(* CODESYS project twincat-tools.library
   Company: hganchev
   DefaultNamespace: tc-tools
   Version: 1.0.0.0
   DocFormat: reStructuredText
   Placeholder: tc-tools
   Author: hganchev
   Title: tc-tools

Project tree, tasks and I/O mapping:
  libraries: Tc2_Standard, * (Beckhoff Automation GmbH); Tc2_System, * (Beckhoff Automation GmbH); Tc2_Utilities, * (Beckhoff Automation GmbH); Tc3_Module, * (Beckhoff Automation GmbH); Tc2_MC2, * (Beckhoff Automation GmbH)
  DUTs/
  GVLs/
    global variables Parameters
  POUs/
    AxisControl/
      function block MC_AxisControl [ST]
    Export/
      function block ExportArrayREALDataToTextFile [ST]
    Range/
      function F_GET_IN_RANGE_INT [ST]
      function F_IN_BOUNDS_ARRAY_INT [ST]
    Round/
      function F_ROUND_LREAL [ST]
      function F_ROUND_REAL [ST]
    String/
      function F_STRING_SPLIT [ST]
    TimeStamp/
      function F_GET_TIME_STAMP [ST]
  Version/
    global variables Global_Version
  VISUs/
*)

// GVLs/Parameters
{attribute 'qualified_only'}
VAR_GLOBAL CONSTANT
	sNewLineSymbol			: STRING(3) := '$0A'; 	// Control character new line, corresponds to '$L' and '$SN'
	sLineBreakSymbol		: STRING(3) := '$0D';	// Control character line break, corresponds to '$R'
	
	// Export Array REAL data to text file parameters
	iArrayREALSize						: INT := 255;
	diByteMultiplierForExport			: DINT := 10; // This multiplies with array Size
	
	// Split Parameters
	iSplitArraySize						: INT := 4;
END_VAR

// Version/Global_Version
{attribute 'TcGenerated'}
{attribute 'no-analysis'}
{attribute 'linkalways'}
// This function has been automatically generated from the project information.
VAR_GLOBAL CONSTANT
	{attribute 'const_non_replaced'}
	stLibVersion_tc_tools : ST_LibVersion := (iMajor := 1, iMinor := 0, iBuild := 0, iRevision := 0, nFlags := 0, sVersion := '1.0.0.0');
END_VAR

// POUs/AxisControl/MC_AxisControl
FUNCTION_BLOCK MC_AxisControl
VAR_INPUT	
END_VAR
VAR_IN_OUT
	axisRef			: AXIS_REF;
END_VAR
VAR_OUTPUT
END_VAR
VAR
	// Controls
	bEnable				: BOOL;
	bHome				: BOOL;
	bReset				: BOOL;
	bMove				: BOOL;
	bStop				: BOOL;
	                	
	// Statuses     	
	bEnabled			: BOOL;
	bReferenced			: BOOL;
	bError				: BOOL;
	nErrorID			: UDINT;
	bMoving				: BOOL;
	bInPosition			: BOOL;
	nActualPosition		: LREAL;
	nActualVelocity		: LREAL;
	
	// Settings
	nTargetPosition		: LREAL;
	nTargetVelocity		: LREAL;
	nTargetAcceleration	: LREAL;
	stHomingOptions		: ST_HomingOptions;
	
	fbEnable			: MC_Power;
	fbHome				: MC_Home;
	fbMove				: MC_MoveAbsolute;
	fbReset				: MC_Reset;
	fbActualPosition	: MC_ReadActualPosition;
	fbActualVelocity	: MC_ReadActualVelocity;
END_VAR

// Power On - power on/off the axis
fbEnable(
	Axis:= axisRef, 
	Enable:= bEnable, 
	Enable_Positive:= bEnable, 
	Enable_Negative:= bEnable, 
	Override:= , 
	BufferMode:= , 
	Options:= , 
	Status=> bEnabled, 
	Busy=> , 
	Active=> , 
	Error=> , 
	ErrorID=> );
	
// Home - Reference the axis
stHomingOptions.ReferenceMode := E_EncoderReferenceMode.ENCODERREFERENCEMODE_DEFAULT;
stHomingOptions.SearchDirection := MC_Direction.MC_Negative_Direction;
stHomingOptions.SearchVelocity := 10;
fbHome(
	Axis:= axisRef, 
	Execute:= bHome AND bEnabled, 
	Position:= 0, 
	HomingMode:= MC_HomingMode.MC_DefaultHoming, 
	BufferMode:= , 
	Options:= stHomingOptions, 
	bCalibrationCam:= , 
	Done=> , 
	Busy=> , 
	Active=> , 
	CommandAborted=> , 
	Error=> , 
	ErrorID=> );
	
// Reset - reset error of axis
fbReset(
	Axis:= axisRef, 
	Execute:= bReset, 
	Done=> , 
	Busy=> , 
	Error=> , 
	ErrorID=> );
	
// Move Absolute - move to absolute position
fbMove(
	Axis:= axisRef, 
	Execute:= bMove AND bEnabled, 
	Position:= nTargetPosition, 
	Velocity:= nTargetVelocity, 
	Acceleration:= nTargetAcceleration, 
	Deceleration:= nTargetAcceleration, 
	Jerk:= , 
	BufferMode:= , 
	Options:= , 
	Done=> , 
	Busy=> , 
	Active=> , 
	CommandAborted=> , 
	Error=> , 
	ErrorID=> );
	
// Status Actual Position
fbActualPosition(
	Axis:= axisRef, 
	Enable:= TRUE, 
	Valid=> , 
	Busy=> , 
	Error=> , 
	ErrorID=> , 
	Position=> nActualPosition);

// Status Actual Velocity	
fbActualVelocity(
	Axis:= axisRef, 
	Enable:= TRUE, 
	Valid=> , 
	Busy=> , 
	Error=> , 
	ErrorID=> , 
	ActualVelocity=> nActualVelocity);
	
// Statuses
axisRef.ReadStatus();
bReferenced := axisRef.Status.Homed;
bMoving := axisRef.Status.Moving;
bInPosition := axisRef.Status.InTargetPosition AND ABS(nTargetPosition - nActualPosition) < 0.1;
bError := axisRef.Status.Error;
nErrorID := axisRef.Status.ErrorID;

// Reset Move
IF bInPosition AND NOT bMoving THEN
	bMove := FALSE;
END_IF

END_FUNCTION_BLOCK

// POUs/Export/ExportArrayREALDataToTextFile
FUNCTION_BLOCK ExportArrayREALDataToTextFile
VAR_INPUT
	arrData 				: ARRAY[0..Parameters.iArrayREALSize] OF REAL;
	bExecute				: BOOL;
	bUseTimeStamp			: BOOL;
	sFilePath				: STRING(255) := 'C:\data.txt';
END_VAR         			
VAR_OUTPUT      			
	bDone					: BOOL;
END_VAR
VAR
	fileOpen				: FB_FileOpen;
//	fileWrite				: FB_FilePuts;
	fileWrite				: FB_FileWrite;
	fileClose				: FB_FileClose;
	                		
	fileHandle				: UINT;
	nSizeWritten			: UDINT;
	
	arrayDataByte			: ARRAY[0..iArrayByteSize] OF BYTE;
	sData					: ARRAY[0..Parameters.iArrayREALSize] OF STRING(255);

	i						: INT;
	j						: INT;
	k						: DINT;	// track of byte array
END_VAR

VAR CONSTANT
	iArrayByteSize 			: DINT := Parameters.diByteMultiplierForExport * Parameters.iArrayREALSize;
END_VAR

bDone := FALSE;
fileClose(bExecute := FALSE);

// file write init
fileWrite(tTimeout:= T#2S);

IF bExecute	THEN	
	// open file
	fileOpen(sPathName := sFilePath, nMode := FOPEN_MODEWRITE,
		 ePath := PATH_GENERIC, hFile => fileHandle, bExecute := TRUE);
		 
	// Clear data
	MEMSET(ADR(arrayDataByte), 16#00, SIZEOF(arrayDataByte));
	
	k := 0;
	// Prepare string data 
	FOR i := 0 TO Parameters.iArrayREALSize DO
		sData[i] := REAL_TO_STRING(arrData[i]);
		IF i > 0 THEN
			sData[i] := CONCAT(Parameters.sNewLineSymbol,sData[i]);
		END_IF
		// Convert to byte for every sData symbol
		FOR j := 0 TO LEN(sData[i]) DO
			MEMCPY(ADR(arrayDataByte[k]),ADR(sData[i][j]), 1);
			k := k + 1;
		END_FOR
	END_FOR
	
	// Write Data
	IF fileHandle <> 0 THEN
		fileWrite(	hFile:= fileHandle, 
					pWriteBuff:= ADR(arrayDataByte), 
					cbWriteLen:= SIZEOF(arrayDataByte), 
					bExecute := TRUE);
	END_IF
	
	IF fileWrite.cbWrite > 0 THEN
		bDone := TRUE;
	END_IF
ELSIF NOT bExecute THEN
	IF NOT fileWrite.bBusy THEN
		fileWrite(bExecute := FALSE);
		fileOpen(bExecute := FALSE);
		fileClose(hFile := fileHandle, bExecute := TRUE);
	END_IF
END_IF

END_FUNCTION_BLOCK

// POUs/Range/F_GET_IN_RANGE_INT
(*
:Info: See <https://github.com/hganchev/twincat-tools/tree/main/TwinCAT%20Tools/twincat-tools/POUs/Range/>
:Author: hganchev <https://github.com/hganchev/>

**Description:**

The F_GET_IN_RANGE_INT function is a custom function in TwinCAT that allows you to map an input integer value from one range to another range.

**Parameters:**

- value (Input): The input integer value that you want to map to the target range.
- range_max (Input): The maximum value of the target range.
- range_min (Input): The minimum value of the target range.
- value_max (Input): The maximum value of the input value range.
- value_min (Input): The minimum value of the input value range.

**Return Value:**

F_GET_IN_RANGE_INT returns an INT value that represents the mapped integer value from the input range to the target range.

**Usage Example:**

.. code::

	VAR
		InputValue : INT := 50;
		MappedValue : INT;
	END_VAR

	// Map InputValue from the range [0, 100] to the range [500, 1000]
	MappedValue := F_GET_IN_RANGE_INT(InputValue, 1000, 500, 100, 0);

In this example, the InputValue variable represents the integer value that you want to map. 
The F_GET_IN_RANGE_INT function is then used to map InputValue from the range [0, 100] to the range [500, 1000]. 
The result is stored in the MappedValue variable.

After executing the code, MappedValue will be equal to 750.
*)
FUNCTION F_GET_IN_RANGE_INT : INT
VAR_INPUT
	value, range_max, range_min, value_max, value_min : INT; // Where range max/min is the range you want to fit the value
END_VAR
VAR
END_VAR

F_GET_IN_RANGE_INT := ((LIMIT(value_min, value, value_max) - value_min)*(range_max - range_min))/(value_max-value_min) + range_min;

END_FUNCTION

// POUs/Range/F_IN_BOUNDS_ARRAY_INT
(*
:Info: See <https://github.com/hganchev/twincat-tools/tree/main/TwinCAT%20Tools/twincat-tools/POUs/Range/>
:Author: hganchev <https://github.com/hganchev/>

**Description:**

The F_IN_BOUNDS_ARRAY_INT function is a custom function in TwinCAT that checks if an index is within the bounds of an integer array.

**Parameters:**

- index (Input): The index to check whether it is within the bounds of the array. 
- arrayIn (Input/Output): The integer array against which the index is checked.

**Return Value:**

F_IN_BOUNDS_ARRAY_INT returns a BOOL value. It is set to TRUE if the index is within the bounds of the array; otherwise, it is set to FALSE.

**Usage Example:**

.. code::

	VAR
		MyArray : ARRAY[1..5] OF INT := [10, 20, 30, 40, 50];
		MyIndex : DINT := 3;
		IsInBounds : BOOL;
	END_VAR
	
	IsInBounds := F_IN_BOUNDS_ARRAY_INT(MyIndex, MyArray);
	
In this example, the MyArray variable represents an integer array with elements [10, 20, 30, 40, 50]. 
The MyIndex variable contains the index that you want to check. 
The F_IN_BOUNDS_ARRAY_INT function is then used to check whether MyIndex is within the bounds of MyArray. 
The result is stored in the IsInBounds variable.

After executing the code, IsInBounds will be set to TRUE since the value of MyIndex (3) is within the bounds of MyArray.
*)

FUNCTION F_IN_BOUNDS_ARRAY_INT : BOOL
VAR_INPUT
	index		: DINT;
END_VAR
VAR_IN_OUT
	arrayIn		: ARRAY[*] OF INT;
END_VAR
VAR
	
END_VAR

F_IN_BOUNDS_ARRAY_INT := index <= UPPER_BOUND(arrayIn, 1) AND index >= LOWER_BOUND(arrayIn, 1);

END_FUNCTION

// POUs/Round/F_ROUND_LREAL
(*
:Info: See <https://github.com/hganchev/twincat-tools/tree/main/TwinCAT%20Tools/twincat-tools/POUs/Round/>
:Author: hganchev <https://github.com/hganchev/>

**Description:**
The F_ROUND_LREAL function is a custom function in TwinCAT that allows you to round a real number to a 
specified number of decimal places.

**Input Parameters:**

- rValue(Input): The lreal number that you want to round.

- iDecNumber(Input): The number of decimal places to round to.

**Return Value:**
F_ROUND_LREAL returns a LREAL value that represents the rounded result of the input number with the specified decimal places.It rounds to higher number if the lef value is bigger or equal than 0.5.

**Usage Example:**

.. code::

	VAR
		MyValue : LREAL := 3.14159;
		RoundedValue : LREAL;
	END_VAR
	
	RoundedValue := F_ROUND_LREAL(MyValue, 2);

In this example, the MyValue variable represents the real number that you want to round. 
The F_ROUND_LREAL function is then used to round MyValue to 2 decimal places. 
The result is stored in the RoundedValue variable.

After executing the code, RoundedValue will contain the rounded value of MyValue with 2 decimal places.
*)
FUNCTION F_ROUND_LREAL : LREAL
VAR_INPUT
	rValue		: LREAL; // Input Value
	iDecNumber	: INT; 	// Numbers after decimal point
END_VAR
VAR
	rOutValue	: LREAL;
	rLeftValue	: LREAL;
END_VAR

rOutValue := rValue * EXPT(10,iDecNumber);
rLeftValue := rOutValue - TRUNC(rOutValue);
IF rLeftValue >= 0.5 THEN
	rOutValue := TRUNC(rOutValue + 1) / EXPT(10,iDecNumber);
ELSIF rLeftValue <= -0.5 THEN
	rOutValue := TRUNC(rOutValue - 1) / EXPT(10,iDecNumber);
ELSE
	rOutValue := TRUNC(rOutValue) / EXPT(10,iDecNumber);
END_IF
F_ROUND_LREAL := rOutValue;

END_FUNCTION

// POUs/Round/F_ROUND_REAL
(*
:Info: See <https://github.com/hganchev/twincat-tools/tree/main/TwinCAT%20Tools/twincat-tools/POUs/Round/>
:Author: hganchev <https://github.com/hganchev/>

**Description:**
The F_ROUND_REAL function is a custom function in TwinCAT that allows you to round a real number to a 
specified number of decimal places.

**Input Parameters:**

- rValue(Input): The real number that you want to round.

- iDecNumber(Input): The number of decimal places to round to.

**Return Value:**
F_ROUND_REAL returns a REAL value that represents the rounded result of the input number with the specified decimal places.It rounds to higher number if the lef value is bigger or equal than 0.5.

**Usage Example:**

.. code::

	VAR
		MyValue : REAL := 3.14159;
		RoundedValue : REAL;
	END_VAR
	
	RoundedValue := F_ROUND_REAL(MyValue, 2);

In this example, the MyValue variable represents the real number that you want to round. 
The F_ROUND_REAL function is then used to round MyValue to 2 decimal places. 
The result is stored in the RoundedValue variable.

After executing the code, RoundedValue will contain the rounded value of MyValue with 2 decimal places.
*)
FUNCTION F_ROUND_REAL : REAL
VAR_INPUT
	rValue		: REAL; // Input Value
	iDecNumber	: INT; 	// Numbers after decimal point
END_VAR
VAR
	rOutValue	: REAL;
	rLeftValue	: REAL;
END_VAR

rOutValue := rValue * EXPT(10,iDecNumber);
rLeftValue := rOutValue - TRUNC(rOutValue);
IF rLeftValue >= 0.5 THEN
	rOutValue := TRUNC(rOutValue + 1) / EXPT(10,iDecNumber);
ELSIF rLeftValue <= -0.5 THEN
	rOutValue := TRUNC(rOutValue - 1) / EXPT(10,iDecNumber);
ELSE
	rOutValue := TRUNC(rOutValue) / EXPT(10,iDecNumber);
END_IF
F_ROUND_REAL := rOutValue;

END_FUNCTION

// POUs/String/F_STRING_SPLIT
(*
:Info: See <https://github.com/hganchev/twincat-tools/tree/main/TwinCAT%20Tools/twincat-tools/POUs/String/>
:Author: hganchev <https://github.com/hganchev/>

**Description:**

This function takes a string sInput and a split character sSplitChar and splits the input string into an array of substrings. 
The resulting array, F_STRING_SPLIT, has a size of Parameters.iSplitArraySize.

**Inputs:**

This function takes a string sInput and a split character sSplitChar and splits the input string into an array of substrings. 
The resulting array, F_STRING_SPLIT, has a size of Parameters.iSplitArraySize.

**Output:**

This implementation iteratively splits the input string using the specified split character. It assigns each substring to the corresponding element in the F_STRING_SPLIT array. 
The splitting process continues until either the end of the input string is reached or the maximum number of substrings specified by Parameters.iSplitArraySize is reached.

**Usage:**

.. code::

	VAR 
		sArray : ARRAY[0..Parameters.iSplitArraySize] OF STRING(255);
	END_VAR
	
	sArray := F_STRING_SPLIT(sInput := 'Hello,World', sSplitChar := ',');
	
Result:

sArray[0] = 'Hello'
sArray[1] = 'World'
*)

FUNCTION F_STRING_SPLIT : ARRAY[0..Parameters.iSplitArraySize] OF STRING(255)
VAR_INPUT
	sInput			: STRING(255);
	sSplitChar		: STRING(1);
END_VAR
VAR
	sCopy			: STRING(255);
	sSplit			: STRING(255);
	iDeleteLen		: INT;
	i				: INT;
END_VAR

sCopy := sInput;

FOR i := 0 TO Parameters.iSplitArraySize DO
	IF FIND(sCopy, sSplitChar) > 0 THEN
		sSplit := LEFT(sCopy, FIND(sCopy, sSplitChar) - 1);
		iDeleteLen := LEN(sSplit) + LEN(sSplitChar);
	ELSE
		sSplit := sCopy;
		iDeleteLen := LEN(sSplit);
	END_IF
	
	// Take the string value
	F_STRING_SPLIT[i] := sSplit;
	
	// Delete 
	sCopy := DELETE(sCopy, iDeleteLen, 1);
	
	// End of split
	IF sCopy = '' THEN
		EXIT;
	END_IF
END_FOR

END_FUNCTION

// POUs/TimeStamp/F_GET_TIME_STAMP
FUNCTION F_GET_TIME_STAMP : STRING(255)
VAR_INPUT
	systemTime				: TIMESTRUCT;			// Using Tc2_Utilities to have the TIMESTRUCT
	strSeparatorDate		: STRING(1) := '_';		// Separator between Year,Month,Day
	strSeparatorTime		: STRING(1) := ':';		// Separator between Hours, Minutes, Seconds		
END_VAR
VAR
	stYear					: STRING;
	stMonth					: STRING;
	stDay					: STRING;
	stHours					: STRING;
	stMinutes				: STRING;
	stSeconds				: STRING;
END_VAR

stYear 		:= CONCAT(WORD_TO_STRING(systemTime.wYear), strSeparatorDate);
stMonth		:= CONCAT(WORD_TO_STRING(systemTime.wMonth), strSeparatorDate);
stDay 		:= CONCAT(WORD_TO_STRING(systemTime.wDay), strSeparatorDate);
stHours 	:= CONCAT(WORD_TO_STRING(systemTime.wHour), strSeparatorTime);
stMinutes 	:= CONCAT(WORD_TO_STRING(systemTime.wMinute), strSeparatorTime);
stSeconds 	:= WORD_TO_STRING(systemTime.wSecond);
F_GET_TIME_STAMP := CONCAT(stYear,CONCAT(stMonth,CONCAT(stDay,CONCAT(stHours,CONCAT(stMinutes,stSeconds)))));

END_FUNCTION
